// TwinCAT 3 PLC project UnitTests2
// ProgramVersion: 3.1.4024.0
// libraries:
//   Tc2_Standard, * (Beckhoff Automation GmbH)
//   Tc2_System, * (Beckhoff Automation GmbH)
//   Tc2_Utilities, * (Beckhoff Automation GmbH)
//   Tc3_Module, * (Beckhoff Automation GmbH)
//   tcl_BaseClasses, * (Red Rock Controls Limited)
//   tcl_StringUtils, * (Red Rock Controls Limited)
//   tcl_UnitTestLibrary, * (Red Rock Controls Limited)
// project tree:
//   GVLs/ GlobalNotifications.TcGVL (not stored)
//   / PlcTask.TcTTO
//   POUs/Assertion/ T_Assertion.TcPOU
//   POUs/ MAIN.TcPOU (not stored)
//   Unit Tests/Execution Result Aggregate/ Test_AggregateResult_Aborted.TcPOU, Test_AggregateResult_Ready.TcPOU, Test_AggregateResult_Busy.TcPOU, Test_AggregateResult_Done.TcPOU, Test_AggregateResult_Error.TcPOU, Test_AggregateResult_ErrorMsg.TcPOU, Test_AggregateResult_Starting.TcPOU, Test_AggregateResult_Aborting.TcPOU
//   Unit Tests/Execution/ Test_TExecutionWhenBusy_Abort_SelectsAborting.TcPOU, Test_TExecutionWhenBusy_SetDone_SetsDone.TcPOU, Test_TExecutionWhenReady_Start_SelectsStarting.TcPOU, Test_TExecution_SetErrorHandlesString_ErrorId.TcPOU
//   Unit Tests/Functions/ Test_ErrorIdToString.TcPOU, Test_F_DINT_TO_UDINT_Conversion.TcPOU, Test_F_Equals.TcPOU, Test_F_NotEqual.TcPOU, Test_F_UDINT_TO_DINT_Conversion.TcPOU
//   Unit Tests/Notifications/ Test_MultipleNotificationsWithStringArgs.TcPOU, Test_NotificationCountWithQueueingEnabled.TcPOU, Test_NotificationHandlerOnlyAddedOnce.TcPOU, Test_NotificationNoArgs.TcPOU, Test_NotificationWithStringArg.TcPOU
//   Unit Tests/ T_TestSuite.TcPOU
// (motion and I/O tree: see PLC project tcl_baseclasses)
// real-time tasks:
//   TASK PlcTask: cycle T#10ms, priority 20, ADS port 350
//   TASK PlcTask1: cycle T#10ms, priority 21, ADS port 351

CONFIGURATION UnitTests2
    RESOURCE PLC ON TwinCAT3
        TASK PlcTask(INTERVAL := T#10ms, PRIORITY := 21);
        PROGRAM MAIN WITH PlcTask : MAIN;
    END_RESOURCE
END_CONFIGURATION

// ---- POUs/Assertion/T_Assertion.TcPOU
FUNCTION_BLOCK T_Assertion
VAR_INPUT
END_VAR
VAR_OUTPUT
END_VAR
VAR
    _AssertionFailed : BOOL;
    _AssertionMessage : T_MaxString;
    _ExpectedAsString : T_MaxString;
    _ActualAsString   : T_MaxString;
END_VAR

METHOD AssertEquals_BOOL : BOOL;
VAR_INPUT
    Source   : T_MaxString;
    Expected : BOOL;
    Actual   : BOOL;
    VariableName : T_MaxString;
END_VAR
AssertEquals_BOOL := AssertTrue(Source    := 'Unit Test',
                                Condition := Expected = Actual,
                                Message   := F_FormatStringEx1('Assertion Failed - %s', VariableName),
                                Failed    =>);
END_METHOD

METHOD AssertEquals_DINT : BOOL
VAR_INPUT
    Source   : T_MaxString;
    Expected : DINT;
    Actual   : DINT;
    VariableName : T_MaxString;
END_VAR
AssertEquals_DINT := AssertTrue(Source    := 'Unit Test',
                                Condition := Expected = Actual,
                                Message   := F_FormatStringEx1('Assertion Failed - %s', VariableName),
                                Failed    =>);
END_METHOD

METHOD AssertEquals_STRING : BOOL
VAR_INPUT
    Source   : T_MaxString;
    Expected : T_MaxString;
    Actual   : T_MaxString;
    VariableName : T_MaxString;
END_VAR
AssertEquals_STRING := AssertTrue(Source    := 'Unit Test',
                                Condition := Expected = Actual,
                                Message   := F_FormatStringEx1('Assertion Failed - %s', VariableName),
                                Failed    =>);
END_METHOD

PROPERTY AssertionFailed : BOOL
GET
AssertionFailed := _AssertionFailed;
END_GET
END_PROPERTY

PROPERTY AssertionMessage : T_MaxString
GET
AssertionMessage := _AssertionMessage;
END_GET
END_PROPERTY

END_FUNCTION_BLOCK

// ---- Unit Tests/Execution Result Aggregate/Test_AggregateResult_Aborted.TcPOU
FUNCTION_BLOCK Test_AggregateResult_Aborted EXTENDS T_UnitTestBase
VAR
    ResultAggregate : T_ResultAggregate;
    Execution1      : T_Execution;
    Execution2      : T_Execution;
    Execution3      : T_Execution;
END_VAR

METHOD Init
Execution1.FB_init(FALSE,FALSE);
Execution2.FB_init(FALSE,FALSE);
Execution3.FB_init(FALSE,FALSE);
END_METHOD

{attribute 'analysis' := '-33'} // inhibit unused variable warning
METHOD RunTest
VAR_OUTPUT
    TestCompleted : BOOL;
    TestFailed    : BOOL;
END_VAR
ResultAggregate.ClearResults();

ResultAggregate.AddResult(Execution1);
ResultAggregate.AddResult(Execution2);
ResultAggregate.AddResult(Execution3);

TestFailed S= NOT AssertFalse(Source    := TestName,
                              Condition := ResultAggregate.Aborted,
                              Message   := 'ResultAggregate.Aborted is not false',
                              Failed    =>);

Execution1.Start();
Execution1.SetBusy();
Execution1.Abort();
Execution1.SetAborted();

Execution2.Start();
Execution2.SetBusy();
Execution2.Abort();
Execution2.SetAborted();

Execution3.Start();
Execution3.SetBusy();
Execution3.Abort();
Execution3.SetAborted();

TestFailed S= NOT AssertTrue(Source    := TestName,
                             Condition := ResultAggregate.Aborted,
                             Message   := 'ResultAggregate.Aborting is false',
                             Failed    =>);

TestCompleted := TRUE;
END_METHOD

END_FUNCTION_BLOCK

// ---- Unit Tests/Execution Result Aggregate/Test_AggregateResult_Ready.TcPOU
FUNCTION_BLOCK Test_AggregateResult_Ready EXTENDS T_UnitTestBase
VAR
    ResultAggregate : T_ResultAggregate;
    Execution1      : T_Execution;
    Execution2      : T_Execution;
    Execution3      : T_Execution;
END_VAR

METHOD Init
Execution1.FB_init(FALSE,FALSE);
Execution2.FB_init(FALSE,FALSE);
Execution3.FB_init(FALSE,FALSE);
END_METHOD

{attribute 'analysis' := '-33'} // inhibit unused variable warning
METHOD RunTest
VAR_OUTPUT
    TestCompleted : BOOL;
    TestFailed    : BOOL;
END_VAR
ResultAggregate.ClearResults();

ResultAggregate.AddResult(Execution1);
ResultAggregate.AddResult(Execution2);
ResultAggregate.AddResult(Execution3);

TestFailed S= NOT AssertTrue(Source    := TestName,
                              Condition := ResultAggregate.Ready,
                              Message   := 'ResultAggregate.Ready is not true',
                              Failed    =>);

Execution1.Start();
Execution1.SetBusy();

TestFailed S= NOT AssertFalse(Source    := TestName,
                             Condition := ResultAggregate.Ready,
                             Message   := 'ResultAggregate.Ready is not false',
                             Failed    =>);

TestCompleted := TRUE;
END_METHOD

END_FUNCTION_BLOCK

// ---- Unit Tests/Execution Result Aggregate/Test_AggregateResult_Busy.TcPOU
FUNCTION_BLOCK Test_AggregateResult_Busy EXTENDS T_UnitTestBase
VAR
	ResultAggregate : T_ResultAggregate;
	Execution1 : T_Execution;
	Execution2 : T_Execution;
	Execution3 : T_Execution;
END_VAR

METHOD Init
Execution1.FB_init(FALSE,FALSE);
Execution2.FB_init(FALSE,FALSE);
Execution3.FB_init(FALSE,FALSE);
END_METHOD

{attribute 'analysis' := '-33'} // inhibit unused variable warning
METHOD RunTest
VAR_OUTPUT
    TestCompleted : BOOL;
    TestFailed    : BOOL;
END_VAR
ResultAggregate.ClearResults();

ResultAggregate.AddResult(Execution1);
ResultAggregate.AddResult(Execution2);
ResultAggregate.AddResult(Execution3);

TestFailed S= NOT AssertFalse(Source    := TestName,
                              Condition := ResultAggregate.Busy,
                              Message   := 'ResultAggregate.Busy is not false',
                              Failed    =>);

Execution1.Start();
Execution1.SetBusy();

TestFailed S= NOT AssertTrue(Source    := TestName,
                             Condition := ResultAggregate.Busy,
                             Message   := 'ResultAggregate.Busy is false',
                             Failed    =>);

TestCompleted := TRUE;
END_METHOD

END_FUNCTION_BLOCK

// ---- Unit Tests/Execution Result Aggregate/Test_AggregateResult_Done.TcPOU
FUNCTION_BLOCK Test_AggregateResult_Done EXTENDS T_UnitTestBase
VAR
	ResultAggregate : T_ResultAggregate;
	Execution1 : T_Execution;
	Execution2 : T_Execution;
	Execution3 : T_Execution;
END_VAR

METHOD Init
Execution1.FB_init(FALSE,FALSE);
Execution2.FB_init(FALSE,FALSE);
Execution3.FB_init(FALSE,FALSE);
END_METHOD

{attribute 'analysis' := '-33'} // inhibit unused variable warning
METHOD RunTest
VAR_OUTPUT
    TestCompleted : BOOL;
    TestFailed    : BOOL;
END_VAR
ResultAggregate.ClearResults();

ResultAggregate.AddResult(Execution1);
ResultAggregate.AddResult(Execution2);
ResultAggregate.AddResult(Execution3);

Execution1.Start();
Execution1.SetBusy();
Execution1.SetDone();

Execution2.Start();
Execution2.SetBusy();
Execution2.SetDone();

TestFailed S= NOT AssertFalse(Source    := TestName,
                              Condition := ResultAggregate.Done,
                              Message   := 'ResultAggregate.Done is not false',
                              Failed    =>);

Execution3.Start();
Execution3.SetBusy();
Execution3.SetDone();

TestFailed S= NOT AssertTrue(Source    := TestName,
                             Condition := ResultAggregate.Done,
                             Message   := 'ResultAggregate.Done is false',
                             Failed    =>);

TestCompleted := TRUE;
END_METHOD

END_FUNCTION_BLOCK

// ---- Unit Tests/Execution Result Aggregate/Test_AggregateResult_Error.TcPOU
FUNCTION_BLOCK Test_AggregateResult_Error EXTENDS T_UnitTestBase
VAR
	ResultAggregate : T_ResultAggregate;
	Execution1 : T_Execution;
	Execution2 : T_Execution;
	Execution3 : T_Execution;
END_VAR

METHOD Init
Execution1.FB_init(FALSE,FALSE);
Execution2.FB_init(FALSE,FALSE);
Execution3.FB_init(FALSE,FALSE);
END_METHOD

{attribute 'analysis' := '-33'} // inhibit unused variable warning
METHOD RunTest
VAR_OUTPUT
    TestCompleted : BOOL;
    TestFailed    : BOOL;
END_VAR
ResultAggregate.ClearResults();

ResultAggregate.AddResult(Execution1);
ResultAggregate.AddResult(Execution2);
ResultAggregate.AddResult(Execution3);

Execution1.Start();
Execution1.SetBusy();

TestFailed S= NOT AssertFalse(Source    := TestName,
                              Condition := ResultAggregate.Error,
                              Message   := 'ResultAggregate.Error is not false',
                              Failed    =>);

Execution3.Start();
Execution3.SetBusy();
Execution3.SetError('Error Message');

TestFailed S= NOT AssertTrue(Source    := TestName,
                             Condition := ResultAggregate.Error,
                             Message   := 'ResultAggregate.Error is false',
                             Failed    =>);

TestCompleted := TRUE;
END_METHOD

END_FUNCTION_BLOCK

// ---- Unit Tests/Execution Result Aggregate/Test_AggregateResult_ErrorMsg.TcPOU
FUNCTION_BLOCK Test_AggregateResult_ErrorMsg EXTENDS T_UnitTestBase
VAR
	ResultAggregate : T_ResultAggregate;
	Execution1 : T_Execution;
	Execution2 : T_Execution;
	Execution3 : T_Execution;
END_VAR

METHOD Init
Execution1.FB_init(FALSE,FALSE);
Execution2.FB_init(FALSE,FALSE);
Execution3.FB_init(FALSE,FALSE);
END_METHOD

{attribute 'analysis' := '-33'} // inhibit unused variable warning
METHOD RunTest
VAR_OUTPUT
    TestCompleted : BOOL;
    TestFailed    : BOOL;
END_VAR
ResultAggregate.ClearResults();

ResultAggregate.AddResult(Execution1);
ResultAggregate.AddResult(Execution2);
ResultAggregate.AddResult(Execution3);

Execution1.Start();
Execution1.SetBusy();
Execution1.SetDone();

Execution2.Start();
Execution2.SetBusy();
Execution2.SetDone();

TestFailed S= NOT AssertTrue(Source    := TestName,
                              Condition := ResultAggregate.ErrorMsg = '',
                              Message   := 'ResultAggregate.ErrorMsg is not blank',
                              Failed    =>);

Execution3.Start();
Execution3.SetBusy();
Execution3.SetError('Error Message');

TestFailed S= NOT AssertTrue(Source    := TestName,
                             Condition := ResultAggregate.ErrorMsg = 'Error Message',
                             Message   := 'ResultAggregate.ErrorMsg is incorrect',
                             Failed    =>);

TestCompleted := TRUE;
END_METHOD

END_FUNCTION_BLOCK

// ---- Unit Tests/Execution Result Aggregate/Test_AggregateResult_Starting.TcPOU
FUNCTION_BLOCK Test_AggregateResult_Starting EXTENDS T_UnitTestBase
VAR
    ResultAggregate : T_ResultAggregate;
    Execution1      : T_Execution;
    Execution2      : T_Execution;
    Execution3      : T_Execution;
END_VAR

METHOD Init
Execution1.FB_init(FALSE,FALSE);
Execution2.FB_init(FALSE,FALSE);
Execution3.FB_init(FALSE,FALSE);
END_METHOD

{attribute 'analysis' := '-33'} // inhibit unused variable warning
METHOD RunTest
VAR_OUTPUT
    TestCompleted : BOOL;
    TestFailed    : BOOL;
END_VAR
ResultAggregate.ClearResults();

ResultAggregate.AddResult(Execution1);
ResultAggregate.AddResult(Execution2);
ResultAggregate.AddResult(Execution3);

TestFailed S= NOT AssertFalse(Source    := TestName,
                              Condition := ResultAggregate.Starting,
                              Message   := 'ResultAggregate.Starting is not false',
                              Failed    =>);

Execution1.Start();

TestFailed S= NOT AssertTrue(Source    := TestName,
                             Condition := ResultAggregate.Starting,
                             Message   := 'ResultAggregate.Starting is false',
                             Failed    =>);

TestCompleted := TRUE;
END_METHOD

END_FUNCTION_BLOCK

// ---- Unit Tests/Execution Result Aggregate/Test_AggregateResult_Aborting.TcPOU
FUNCTION_BLOCK Test_AggregateResult_Aborting EXTENDS T_UnitTestBase
VAR
    ResultAggregate : T_ResultAggregate;
    Execution1      : T_Execution;
    Execution2      : T_Execution;
    Execution3      : T_Execution;
END_VAR

METHOD Init
Execution1.FB_init(FALSE,FALSE);
Execution2.FB_init(FALSE,FALSE);
Execution3.FB_init(FALSE,FALSE);
END_METHOD

{attribute 'analysis' := '-33'} // inhibit unused variable warning
METHOD RunTest
VAR_OUTPUT
    TestCompleted : BOOL;
    TestFailed    : BOOL;
END_VAR
ResultAggregate.ClearResults();

ResultAggregate.AddResult(Execution1);
ResultAggregate.AddResult(Execution2);
ResultAggregate.AddResult(Execution3);

TestFailed S= NOT AssertFalse(Source    := TestName,
                              Condition := ResultAggregate.Aborting,
                              Message   := 'ResultAggregate.Aborting is not false',
                              Failed    =>);

Execution3.Start();
Execution3.SetBusy();
Execution3.Abort();

TestFailed S= NOT AssertTrue(Source    := TestName,
                             Condition := ResultAggregate.Aborting,
                             Message   := 'ResultAggregate.Aborting is false',
                             Failed    =>);

TestCompleted := TRUE;
END_METHOD

END_FUNCTION_BLOCK

// ---- Unit Tests/Execution/Test_TExecutionWhenBusy_Abort_SelectsAborting.TcPOU
FUNCTION_BLOCK Test_TExecutionWhenBusy_Abort_SelectsAborting EXTENDS T_UnitTestbase
VAR
    Execution : T_Execution;
END_VAR

METHOD Init
Execution.FB_init(bInitRetains := FALSE,
                  bInCopyCode  := FALSE);
END_METHOD

{attribute 'analysis' := '-33'} // inhibit unused variable warning
METHOD RunTest
VAR_OUTPUT
    TestCompleted : BOOL;
    TestFailed    : BOOL;
END_VAR
Execution.Start();
Execution.SetBusy();
Execution.Abort();

TestFailed S= NOT AssertTrue(Source    := TestName,
                             Condition := Execution.Aborting,
                             Message   := 'Execution.Aborting not true');

TestCompleted := TRUE;
END_METHOD

END_FUNCTION_BLOCK

// ---- Unit Tests/Execution/Test_TExecutionWhenBusy_SetDone_SetsDone.TcPOU
FUNCTION_BLOCK Test_TExecutionWhenBusy_SetDone_SetsDone EXTENDS T_UnitTestbase
VAR
    Execution : T_Execution;
END_VAR

METHOD Init
// Setup...
Execution.FB_init(bInitRetains := FALSE,
                  bInCopyCode  := FALSE);
END_METHOD

{attribute 'analysis' := '-33'} // inhibit unused variable warning
METHOD RunTest
VAR_OUTPUT
    TestCompleted : BOOL;
    TestFailed    : BOOL;
END_VAR
// Test...
Execution.Start();
Execution.SetBusy();
Execution.SetDone();
					
TestFailed S= NOT AssertTrue(Source    := TestName,
                             Condition := Execution.Done,
                             Message   := 'Execution.Done not true');

TestFailed S= NOT AssertTrue(Source    := TestName,
                             Condition := Execution.Ready,
                             Message   := 'Execution.Ready not true');

TestCompleted := TRUE;
END_METHOD

END_FUNCTION_BLOCK

// ---- Unit Tests/Execution/Test_TExecutionWhenReady_Start_SelectsStarting.TcPOU
FUNCTION_BLOCK Test_TExecutionWhenReady_Start_SelectsStarting EXTENDS T_UnitTestbase
VAR
    Execution : T_Execution;
END_VAR

METHOD Init
// Setup...
Execution.FB_init(bInitRetains := FALSE,
                  bInCopyCode  := FALSE);
END_METHOD

{attribute 'analysis' := '-33'} // inhibit unused variable warning
METHOD RunTest
VAR_OUTPUT
    TestCompleted : BOOL;
    TestFailed    : BOOL;
END_VAR
// Test...
Execution.Start();

TestFailed S= NOT AssertTrue(Source    := TestName,
                             Condition := Execution.Starting,
                             Message   := 'Execution.Starting not true');

TestCompleted := TRUE;
END_METHOD

END_FUNCTION_BLOCK

// ---- Unit Tests/Execution/Test_TExecution_SetErrorHandlesString_ErrorId.TcPOU
FUNCTION_BLOCK Test_TExecution_SetErrorHandlesString_ErrorId EXTENDS T_UnitTestBase
VAR
    Execution : T_Execution;
END_VAR
VAR
    ErrorId : STRING := 'Custom error message';
END_VAR

METHOD Init
END_METHOD

{attribute 'analysis' := '-33'} // inhibit unused variable warning
METHOD RunTest
VAR_OUTPUT
    TestCompleted : BOOL;
    TestFailed    : BOOL;
END_VAR
VAR
    ErrorMsg : STRING := 'Custom error message';
END_VAR
Execution.Start();
Execution.SetBusy();
Execution.SetError(ErrorMsg);

TestFailed S= NOT AssertTrue(Source    := TestName,
                             Condition := Execution.ErrorMsg = 'Custom error message',
                             Message   := 'Execution.ErrorMsg not correct');

TestCompleted := TRUE;
END_METHOD

END_FUNCTION_BLOCK

// ---- Unit Tests/Functions/Test_ErrorIdToString.TcPOU
FUNCTION_BLOCK Test_ErrorIdToString EXTENDS T_UnitTestBase
VAR_INPUT
END_VAR
VAR_OUTPUT
END_VAR
VAR
	Assertion : T_Assertion;
END_VAR

{attribute 'analysis' := '-33'} // inhibit unused variable warning
METHOD RunTest
VAR_OUTPUT
    TestCompleted : BOOL;
    TestFailed    : BOOL;
END_VAR
TestFailed S= NOT Assertion.AssertEquals_STRING(Source    := TestName,
                             Expected     := 'Error 0x12BD',
                              Actual       := F_ErrorIdToString(16#12BD),
                              VariableName := 'F_ErrorIdToString(16#12BD)');

TestFailed S= NOT Assertion.AssertEquals_STRING(Source    := TestName,
                             Expected     := 'Error 0x12345678',
                              Actual       := F_ErrorIdToString(16#12345678),
                              VariableName := 'F_ErrorIdToString(16#12345678)');

TestFailed S= NOT Assertion.AssertEquals_STRING(Source    := TestName,
                             Expected     := 'Error 0x00FF',
                              Actual       := F_ErrorIdToString(16#FF),
                              VariableName := 'F_ErrorIdToString(16#FF)');

TestFailed S= NOT Assertion.AssertEquals_STRING(Source    := TestName,
                             Expected     := 'Error 0x0011 - No debugging available',
                              Actual       := F_ErrorIdToString(16#11),
                              VariableName := 'F_ErrorIdToString(16#11)');

TestCompleted := TRUE;
END_METHOD

END_FUNCTION_BLOCK

// ---- Unit Tests/Functions/Test_F_DINT_TO_UDINT_Conversion.TcPOU
FUNCTION_BLOCK Test_F_DINT_TO_UDINT_Conversion EXTENDS T_UnitTestBase
VAR
    InputValue     : DINT;
    ConvertedValue : UDINT;
	Assertion : T_Assertion;
END_VAR

{attribute 'analysis' := '-33'} // inhibit unused variable warning
METHOD RunTest
VAR_OUTPUT
    TestCompleted : BOOL;
    TestFailed    : BOOL;
END_VAR
InputValue     := 2147483648;                  // too big
ConvertedValue := F_UDINT_TO_DINT(InputValue); // limit to largest DINT

TestFailed S= NOT Assertion.AssertEquals_DINT(Source    := TestName,
                             Expected     := 2147483647,
                            Actual       := ConvertedValue,
                            VariableName := 'ConvertedValue');

TestCompleted := TRUE;
END_METHOD

END_FUNCTION_BLOCK

// ---- Unit Tests/Functions/Test_F_Equals.TcPOU
FUNCTION_BLOCK Test_F_Equals EXTENDS T_UnitTestBase
VAR
	Assertion : T_Assertion;
END_VAR

{attribute 'analysis' := '-33'} // inhibit unused variable warning
METHOD RunTest
VAR_OUTPUT
    TestCompleted : BOOL;
    TestFailed    : BOOL;
END_VAR
TestFailed S= NOT Assertion.AssertEquals_BOOL(Source    := TestName,
                             Expected := TRUE,
                            Actual   := F_Equals(1.000_005,
                                                 1.000_004,
                                                 0.000_002),
                            VariableName := 'F_Equals');

TestFailed S= NOT Assertion.AssertEquals_BOOL(Source    := TestName,
                             Expected := FALSE,
                            Actual   := F_Equals(1.000_005,
                                                 1.000_003,
                                                 0.000_001),
                            VariableName := 'F_Equals');

TestCompleted := TRUE;
END_METHOD

END_FUNCTION_BLOCK

// ---- Unit Tests/Functions/Test_F_NotEqual.TcPOU
FUNCTION_BLOCK Test_F_NotEqual EXTENDS T_UnitTestBase
VAR
	Assertion : T_Assertion;
END_VAR

{attribute 'analysis' := '-33'} // inhibit unused variable warning
METHOD RunTest
VAR_OUTPUT
    TestCompleted : BOOL;
    TestFailed    : BOOL;
END_VAR
TestFailed S= NOT Assertion.AssertEquals_BOOL(Source    := TestName,
                             Expected := TRUE,
                            Actual   := F_NotEqual(1.000_005,
                                                   1.000_003,
                                                   0.000_001),
                            VariableName := 'F_Equals');

TestFailed S= NOT Assertion.AssertEquals_BOOL(Source    := TestName,
                             Expected := FALSE,
                            Actual   := F_NotEqual(1.000_005,
                                                   1.000_004,
                                                   0.000_002),
                            VariableName := 'F_Equals');

TestCompleted := TRUE;
END_METHOD

END_FUNCTION_BLOCK

// ---- Unit Tests/Functions/Test_F_UDINT_TO_DINT_Conversion.TcPOU
FUNCTION_BLOCK Test_F_UDINT_TO_DINT_Conversion EXTENDS T_UnitTestBase
VAR
    InputValue     : UDINT;
    ConvertedValue : DINT;
	Assertion : T_Assertion;
END_VAR

{attribute 'analysis' := '-33'} // inhibit unused variable warning
METHOD RunTest
VAR_OUTPUT
    TestCompleted : BOOL;
    TestFailed    : BOOL;
END_VAR
InputValue     := 2147483648;                  // too big
ConvertedValue := F_UDINT_TO_DINT(InputValue); // limit to largest DINT

TestFailed S= NOT Assertion.AssertEquals_DINT(Source    := TestName,
                             Expected     := 2147483647,
                            Actual       := ConvertedValue,
                            VariableName := 'ConvertedValue');

TestCompleted := TRUE;
END_METHOD

END_FUNCTION_BLOCK

// ---- Unit Tests/Notifications/Test_MultipleNotificationsWithStringArgs.TcPOU
{attribute 'hide'}
FUNCTION_BLOCK Test_MultipleNotificationsWithStringArgs EXTENDS T_UnitTestBase
VAR
    Source  : T_Notification;
    Handler : T_NotificationHandler;

    IsRaised          : BOOL;
    NotificationCount : DINT;
	Assertion : T_Assertion;
END_VAR

{attribute 'analysis' := '-33'} // inhibit unused variable warning
METHOD RunTest
VAR_OUTPUT
    TestCompleted : BOOL;
    TestFailed    : BOOL;
END_VAR
Handler.FB_init(bInitRetains := FALSE,
                bInCopyCode  := FALSE);

IsRaised          := FALSE;
NotificationCount := 0;

Source.ClearNotificationHandlers().AddNotificationHandler(Handler);
Source.Args.Init(8);

Source.Args.Clear()
    .Add_INT(1234).Add_STRING('String1');

Source.Raise();

Source.Args.Clear()
    .Add_INT(5678).Add_STRING('String2');

Source.Raise();

TestFailed S= NOT Assertion.AssertEquals_DINT(Source    := TestName,
                             Expected     := 2,
                            Actual       := Handler.NotificationCount,
                            VariableName := 'Handler.NotificationCount');

TestFailed S= NOT Assertion.AssertEquals_BOOL(Source    := TestName,
                             Expected     := TRUE,
                            Actual       := Handler.IsRaised(),
                            VariableName := 'Handler.IsRaised()');

TestFailed S= NOT Assertion.AssertEquals_DINT(Source    := TestName,
                             Expected     := 1,
                            Actual       := Handler.NotificationCount,
                            VariableName := 'Handler.NotificationCount');

TestFailed S= NOT Assertion.AssertEquals_DINT(Source    := TestName,
                             Expected     := 1234,
                            Actual       := Handler.Args.Read_INT(),
                            VariableName := 'Handler.Args.Read_INT()');

TestFailed S= NOT Assertion.AssertEquals_STRING(Source    := TestName,
                             Expected     := 'String1',
                              Actual       := Handler.Args.Read_STRING(),
                              VariableName := 'Handler.Args.Read_STRING()');

TestFailed S= NOT Assertion.AssertEquals_BOOL(Source    := TestName,
                             Expected     := TRUE,
                            Actual       := Handler.IsRaised(),
                            VariableName := 'Handler.IsRaised()');

TestFailed S= NOT Assertion.AssertEquals_DINT(Source    := TestName,
                             Expected     := 0,
                            Actual       := Handler.NotificationCount,
                            VariableName := 'Handler.NotificationCount');

TestFailed S= NOT Assertion.AssertEquals_DINT(Source    := TestName,
                             Expected     := 5678,
                            Actual       := Handler.Args.Read_INT(),
                            VariableName := 'Handler.Args.Read_INT()');

TestFailed S= NOT Assertion.AssertEquals_STRING(Source    := TestName,
                             Expected     := 'String2',
                              Actual       := Handler.Args.Read_STRING(),
                              VariableName := 'Handler.Args.Read_STRING()');

TestFailed S= NOT Assertion.AssertEquals_BOOL(Source    := TestName,
                             Expected     := FALSE,
                            Actual       := Handler.IsRaised(),
                            VariableName := 'Handler.IsRaised()');

TestCompleted := TRUE;
END_METHOD

END_FUNCTION_BLOCK

// ---- Unit Tests/Notifications/Test_NotificationCountWithQueueingEnabled.TcPOU
FUNCTION_BLOCK Test_NotificationCountWithQueueingEnabled EXTENDS T_UnitTestBase
VAR
    Notification   : T_Notification;
    NotificationHandler : T_NotificationHandler;
    IsRaised : BOOL;
	Assertion : T_Assertion;
END_VAR

{attribute 'analysis' := '-33'} // inhibit unused variable warning
METHOD RunTest
VAR_OUTPUT
    TestCompleted : BOOL;
    TestFailed    : BOOL;
END_VAR
NotificationHandler.FB_init(bInitRetains    := FALSE,
                            bInCopyCode     := FALSE);
							
NotificationHandler.NotificationQueueingEnabled := TRUE; // Notification Queuing requires care to ensure all notifications are handled, so disabled by default!

Notification.ClearNotificationHandlers().AddNotificationHandler(NotificationHandler);

Notification.Raise();
Notification.Raise();
Notification.Raise();

TestFailed S= NOT Assertion.AssertEquals_DINT(Source       := TestName,
                                              Expected     := 3,
                                              Actual       := NotificationHandler.NotificationCount,
                                              VariableName := 'Handler.NotificationCount');

TestFailed S= NOT Assertion.AssertEquals_BOOL(Source       := TestName,
                                              Expected     := TRUE,
                                              Actual       := NotificationHandler.IsRaised(),
                                              VariableName := 'IsRaised');

TestFailed S= NOT Assertion.AssertEquals_DINT(Source       := TestName,
                                              Expected     := 2,
                                              Actual       := NotificationHandler.NotificationCount,
                                              VariableName := 'Handler.NotificationCount');

TestFailed S= NOT Assertion.AssertEquals_BOOL(Source       := TestName,
                                              Expected     := TRUE,
                                              Actual       := NotificationHandler.IsRaised(),
                                              VariableName := 'IsRaised');

TestFailed S= NOT Assertion.AssertEquals_DINT(Source       := TestName,
                                              Expected     := 1,
                                              Actual       := NotificationHandler.NotificationCount,
                                              VariableName := 'Handler.NotificationCount');

IsRaised   := NotificationHandler.IsRaised();
TestFailed S= NOT Assertion.AssertEquals_BOOL(Source       := TestName,
                                              Expected     := TRUE,
                                              Actual       := IsRaised,
                                              VariableName := 'IsRaised');

TestFailed S= NOT Assertion.AssertEquals_DINT(Source       := TestName,
                                              Expected     := 0,
                                              Actual       := NotificationHandler.NotificationCount,
                                              VariableName := 'Handler.NotificationCount');

TestFailed S= NOT Assertion.AssertEquals_BOOL(Source       := TestName,
                                              Expected     := FALSE,
                                              Actual       := NotificationHandler.IsRaised(),
                                              VariableName := 'Handler.IsRaised()');

TestCompleted := TRUE;
END_METHOD

END_FUNCTION_BLOCK

// ---- Unit Tests/Notifications/Test_NotificationHandlerOnlyAddedOnce.TcPOU
FUNCTION_BLOCK Test_NotificationHandlerOnlyAddedOnce EXTENDS T_UnitTestBase
VAR
    Notification        : T_Notification;
    NotificationHandler : T_NotificationHandler;
    IsRaised            : BOOL;
    Assertion           : T_Assertion;
END_VAR

{attribute 'analysis' := '-33'} // inhibit unused variable warning
METHOD RunTest
VAR_OUTPUT
    TestCompleted : BOOL;
    TestFailed    : BOOL;
END_VAR
NotificationHandler.FB_init(bInitRetains := FALSE,
                            bInCopyCode     := FALSE);

Notification
	.ClearNotificationHandlers()
	.AddNotificationHandler(NotificationHandler)
	.AddNotificationHandler(NotificationHandler);

Notification.Raise();
IsRaised := NotificationHandler.IsRaised();

TestFailed S= NOT Assertion.AssertEquals_BOOL(Source    := TestName,
                             Expected     := TRUE,
                            Actual       := IsRaised,
                            VariableName := 'IsRaised');

IsRaised := NotificationHandler.IsRaised();

TestFailed S= NOT Assertion.AssertEquals_BOOL(Source    := TestName,
                             Expected     := FALSE,
                            Actual       := IsRaised,
                            VariableName := 'IsRaised');

TestCompleted := TRUE;
END_METHOD

END_FUNCTION_BLOCK

// ---- Unit Tests/Notifications/Test_NotificationNoArgs.TcPOU
FUNCTION_BLOCK Test_NotificationNoArgs EXTENDS T_UnitTestBase
VAR
    Notification        : T_Notification;
    NotificationHandler : T_NotificationHandler;
    IsRaised            : BOOL;
    Assertion           : T_Assertion;
END_VAR

{attribute 'analysis' := '-33'} // inhibit unused variable warning
METHOD RunTest
VAR_OUTPUT
    TestCompleted : BOOL;
    TestFailed    : BOOL;
END_VAR
NotificationHandler.FB_init(bInitRetains    := FALSE,
                            bInCopyCode     := FALSE);

Notification.ClearNotificationHandlers().AddNotificationHandler(NotificationHandler);

Notification.Raise();
IsRaised := NotificationHandler.IsRaised();

TestFailed S= NOT Assertion.AssertEquals_BOOL(Source       := TestName,
                                              Expected     := TRUE,
                                              Actual       := IsRaised,
                                              VariableName := 'IsRaised');

TestCompleted := TRUE;
END_METHOD

END_FUNCTION_BLOCK

// ---- Unit Tests/Notifications/Test_NotificationWithStringArg.TcPOU
{attribute 'hide'}
FUNCTION_BLOCK Test_NotificationWithStringArg EXTENDS T_UnitTestBase
VAR
    Notification        : T_Notification;
    NotificationHandler : T_NotificationHandler;

    ResultString : T_MaxString;
    Args         : I_StreamReader;
    IsRaised     : BOOL;
    Assertion    : T_Assertion;
END_VAR

{attribute 'analysis' := '-33'} // inhibit unused variable warning
METHOD RunTest
VAR_OUTPUT
    TestCompleted : BOOL;
    TestFailed    : BOOL;
END_VAR
NotificationHandler.FB_init(bInitRetains    := FALSE,
                            bInCopyCode     := FALSE);

Notification.ClearNotificationHandlers().AddNotificationHandler(NotificationHandler);
Notification.Args.Init(81);

Notification.Args.Clear().Add_STRING('Big long string passed to the notification handler for later use');
Notification.Raise();

IF NotificationHandler.IsRaised() THEN
    Args         := NotificationHandler.Args;
    ResultString := Args.Read_STRING();
END_IF

TestFailed S= NOT Assertion.AssertEquals_STRING(Source       := TestName,
                                                Expected     := 'Big long string passed to the notification handler for later use',
                                                Actual       := ResultString,
                                                VariableName := 'ResultString');

TestCompleted := TRUE;
END_METHOD

END_FUNCTION_BLOCK

// ---- Unit Tests/T_TestSuite.TcPOU
FUNCTION_BLOCK T_TestSuite
VAR
    TestRunner : T_TestRunner(TestSuiteName    := 'tcl_BaseClasses Tests',
                              Verbose          := TRUE,
                              StopOnFailedTest := TRUE,
                              RunOnDownload    := TRUE);

    Test_AggregateResult_Ready    : Test_AggregateResult_Ready(TestRunner);
    Test_AggregateResult_Starting : Test_AggregateResult_Starting(TestRunner);
    Test_AggregateResult_Busy     : Test_AggregateResult_Busy(TestRunner);
    Test_AggregateResult_Done     : Test_AggregateResult_Done(TestRunner);
    Test_AggregateResult_Error    : Test_AggregateResult_Error(TestRunner);
    Test_AggregateResult_ErrorMsg : Test_AggregateResult_ErrorMsg(TestRunner);
    Test_AggregateResult_Aborting : Test_AggregateResult_Aborting(TestRunner);
    Test_AggregateResult_Aborted  : Test_AggregateResult_Aborted(TestRunner);

    Test_TExecution_WhenBusy_Abort_SelectsAborting  : Test_TExecutionWhenBusy_Abort_SelectsAborting(TestRunner);
    Test_TExecution_WhenBusy_SetDone_SetsDone       : Test_TExecutionWhenBusy_SetDone_SetsDone(TestRunner);
    Test_TExecution_WhenReady_Start_SelectsStarting : Test_TExecutionWhenReady_Start_SelectsStarting(TestRunner);
    Test_TExecution_SetErrorHandlesString_ErrorId   : Test_TExecution_SetErrorHandlesString_ErrorId(TestRunner);

    Test_F_DINT_TO_UDINT_Conversion : Test_F_DINT_TO_UDINT_Conversion(TestRunner);
    Test_F_UDINT_TO_DINT_Conversion : Test_F_UDINT_TO_DINT_Conversion(TestRunner);
    Test_F_Equals                   : Test_F_Equals(TestRunner);
    Test_F_NotEqual                 : Test_F_NotEqual(TestRunner);
    Test_ErrorIdToString            : Test_ErrorIdToString(TestRunner);

    Test_NotificationNoArgs                   : Test_NotificationNoArgs(TestRunner);
    Test_NotificationWithStringArg            : Test_NotificationWithStringArg(TestRunner);
    Test_NotificationCountWithQueueingEnabled : Test_NotificationCountWithQueueingEnabled(TestRunner);
    Test_MultipleNotificationsWithStringArgs  : Test_MultipleNotificationsWithStringArgs(TestRunner);
    Test_NotificationHandlerOnlyAddedOnce     : Test_NotificationHandlerOnlyAddedOnce(TestRunner);
END_VAR

TestRunner.CyclicUpdate();

END_FUNCTION_BLOCK
